FUNCTION_BLOCK Button
VAR
	_input	: BOOL;
END_VAR

PROPERTY IsPressed : BOOL
GET
IsPressed:= _input;
END_GET
END_PROPERTY

END_FUNCTION_BLOCK

(* stored: Version 1.1.0.1, ProductVersion 3.1.4024.12
   POU Button: Id {310a0ffc-7dae-4cca-bf93-4d4c96def001}, SpecialFunc None
   Property IsPressed: Id {b362d482-2d17-4a5d-ba41-a7011dc106a1}
   Get Get: Id {a0cc68e7-5a00-4b3c-846d-23a34c93bfe8} *)
